INTERFACE I_Configuration_Station

METHOD Check : BOOL
END_METHOD

METHOD PRIVATE Cmd : E_DATA_STATE
VAR_INPUT
  Ctrl      : E_DATA_CTRL;
END_VAR
END_METHOD

PROPERTY Ctrl : REFERENCE to ST_DATA_CTRL
SET
END_SET
END_PROPERTY

PROPERTY Identity : OTCID
GET
END_GET
SET
END_SET
END_PROPERTY

PROPERTY State : REFERENCE TO ST_DATA_STATE
SET
END_SET
END_PROPERTY

PROPERTY StationParameter : pointer to ARRAY[1..MAX_STATION] OF ST_STATION_PARAMETER
SET
END_SET
END_PROPERTY

END_INTERFACE

(* stored: Version 1.1.0.1
   Itf I_Configuration_Station: Id {e09684d4-20f8-4435-abdd-440adcf34e07}
   Folder methods: Id {9148e9ec-fdd6-48a6-a52f-1ddf79ce5319}
   Folder properties: Id {27e80ced-1240-4cc1-b0e0-6bb39bbbd653}
   Method Check: Id {671bf40f-c6e5-450c-8a05-e92117b8be6c}
   Method Cmd: Id {32fae96c-b3d7-4f29-88e7-ecfeb58c4f4e}
   Property Ctrl: Id {0595a3b5-09de-4f23-b0a0-0e5d22a714bf}
   Set Set: Id {33612383-b171-4f25-a41c-f7988d29c9ba}
   Property Identity: Id {a5ea37e9-4bf9-4469-a87d-4e7d89f9b631}
   Get Get: Id {7d8960df-747c-46fe-955b-a1b328c38488}
   Set Set: Id {5b4c65a5-0042-496f-be99-9e5d6ea7c5b2}
   Property State: Id {069e82c5-b3ac-42d6-ba50-bf2bc3906046}
   Set Set: Id {af2c795f-b287-488a-8030-161b4ed41c32}
   Property StationParameter: Id {ff8cdaae-a85a-4003-b701-6f0c34435c16}
   Set Set: Id {87290c11-464a-4f36-b13b-d8f4e7360029} *)
